// TIA Portal V20 export
FUNCTION "LER_SimHmiLinearAxis" : Void   // FC36, LAD
// stored: Access Published, IsIECCheckEnabled true, SetENOAutomatically true
   VAR_INPUT
      hmiMode : Int;   // 1:L2R Large, 2:L2R Samll, 3:R2L Large, 4:R2L Small
      hmiMinLimit : LReal;   // TO_Software Min Limit
      hmiMaxLimit : LReal;   // TO_Software Max Limit
      axisActualPos : LReal;
      referenceDesignator : WString;
   END_VAR
   VAR_OUTPUT
      simHmiAxis : "LER_typeSimLinearAxis";
   END_VAR
   VAR_TEMP
      t_ratio : LReal;
      t_axisTravelDistance : LReal;
      t_hmiPositionLReal : LReal;
      t_hmiTravleDistance : Int;
   END_VAR
   VAR CONSTANT
      L2R_LARGE_MIN_PIXEL : Int := 72;
      L2R_LARGE_MAX_PIXEL : Int := 632;
      L2R_SMALL_MIN_PIXEL : Int := 72;
      L2R_SMALL_MAX_PIXEL : Int := 192;
      R2L_LARGE_MIN_PIXEL : Int := 0;
      R2L_LARGE_MAX_PIXEL : Int := 560;
      R2L_SMALL_MIN_PIXEL : Int := 0;
      R2L_SMALL_MAX_PIXEL : Int := 120;
   END_VAR
BEGIN

REGION Network 1 (SCL): i_mode == 1 // L2R Large

   IF #hmiMode = 1 THEN
     #t_hmiTravleDistance := #L2R_LARGE_MAX_PIXEL - #L2R_LARGE_MIN_PIXEL;
     #t_axisTravelDistance := #hmiMaxLimit - #hmiMinLimit;
     #t_ratio := (#axisActualPos - #hmiMinLimit) / #t_axisTravelDistance;

     #simHmiAxis.hmiObjectPos := #L2R_LARGE_MIN_PIXEL + LREAL_TO_INT((#t_ratio * INT_TO_LREAL(#t_hmiTravleDistance)));

   END_IF;
END_REGION

REGION Network 2 (SCL): i_mode == 2 // L2R Small

   IF #hmiMode = 2 THEN
     #t_hmiTravleDistance := #L2R_SMALL_MAX_PIXEL - #L2R_SMALL_MIN_PIXEL;
     #t_axisTravelDistance := #hmiMaxLimit - #hmiMinLimit;
     #t_ratio := (#axisActualPos - #hmiMinLimit) / #t_axisTravelDistance;

     #simHmiAxis.hmiObjectPos := #L2R_SMALL_MIN_PIXEL + LREAL_TO_INT((#t_ratio * INT_TO_LREAL(#t_hmiTravleDistance)));

   END_IF;
END_REGION

REGION Network 3 (SCL): i_mode == 3 // R2L Large

   IF #hmiMode = 3 THEN
     #t_hmiTravleDistance := #R2L_LARGE_MAX_PIXEL - #R2L_LARGE_MIN_PIXEL;
     #t_axisTravelDistance := #hmiMaxLimit - #hmiMinLimit;
     #t_ratio := (#axisActualPos - #hmiMinLimit) / #t_axisTravelDistance;

     #simHmiAxis.hmiObjectPos := #R2L_LARGE_MAX_PIXEL - LREAL_TO_INT((#t_ratio * INT_TO_LREAL(#t_hmiTravleDistance)));

   END_IF;
END_REGION

REGION Network 4 (SCL): i_mode == 4 // R2L Small

   IF #hmiMode = 4 THEN
     #t_hmiTravleDistance := #R2L_SMALL_MAX_PIXEL - #R2L_SMALL_MIN_PIXEL;
     #t_axisTravelDistance := #hmiMaxLimit - #hmiMinLimit;
     #t_ratio := (#axisActualPos - #hmiMinLimit) / #t_axisTravelDistance;

     #simHmiAxis.hmiObjectPos := #R2L_SMALL_MAX_PIXEL - LREAL_TO_INT((#t_ratio * INT_TO_LREAL(#t_hmiTravleDistance)));

   END_IF;
END_REGION

REGION Network 5: Output Mapping
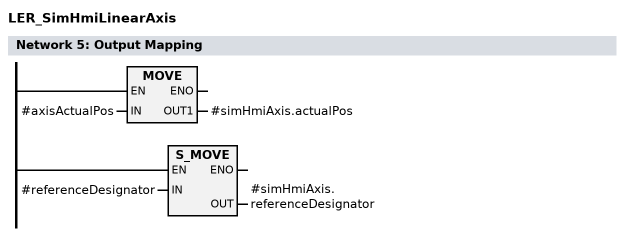
   RUNG wire#powerrail
      Move(in := #axisActualPos, out1 => #simHmiAxis.actualPos)
   END_RUNG
   RUNG wire#powerrail
      S_Move(in := #referenceDesignator, out => #simHmiAxis.referenceDesignator)
   END_RUNG
   // the same network as SCL:
   #simHmiAxis.actualPos := #axisActualPos;
   #simHmiAxis.referenceDesignator := #referenceDesignator;
END_REGION
END_FUNCTION
